// TIA Portal V20 export
DATA_BLOCK "DB_Impulsion"   // DB84
// stored: InstanceOfName FB_Impulsion, InstanceOfType FB
"FB_Impulsion"
   // VAR RETAIN
   //    sCountSecPulseMinute : DInt;
   //    sCountSecPulseHour : DInt;
   //    sCountSecPulseDay : DInt;
   // END_VAR
   // VAR
   //    sPulseMinute : Bool;
   //    sPulseHour : Bool;
   //    sPulseDay : Bool;
   //    sRT_Clock_1Hz { S7_SetPoint := 'True'} : R_TRIG;
   // END_VAR
BEGIN
END_DATA_BLOCK
